FUNCTION_BLOCK FB_EP7402_Scan_Motor
VAR CONSTANT
	cnValueChannel_1: UINT:=16#8007;
	cnValueChannel_2: UINT:=16#8017;
END_VAR
VAR_INPUT
	bExecute:BOOL;
	sNetId 		: T_AmsNetID;
	tUpdateInterval:TIME:=T#1S;
	nSlaveAddr	: UINT;
	bMotorChannel_1:BOOL:= TRUE;
END_VAR
VAR_OUTPUT
	bBusy:BOOL;
	nProgress: USINT;
	aResponse:ARRAY [1..6] OF BYTE;
	bError:BOOL;
	nErrId:UDINT;
END_VAR
VAR
	fbWriteCoEParameter	:  FB_EcCoESdoWrite;
	fbReadCoEParameter	:  FB_EcCoESdoRead;
	fbReadCoEParameterEx	:  FB_EcCoESdoReadEx;
	fbRequestProgress:f_trig;
	nStep:(init, request_command_register, requesting_command_register ,send_request, sending_request, request_progress, requesting_progress, request_error, requesting_error);
	fbExecuteTrigger:r_trig;
	nStatus:USINT;
	aBuffer: array [1..12] of Byte;
	
END_VAR

fbExecuteTrigger(clk:=bExecute);
IF fbExecuteTrigger.q THEN
	nStep:=request_command_register;
	nProgress:=0;
	memset(ADR(aResponse),0,SIZEOF(aResponse));
	bBusy:=TRUE;
END_IF



CASE nStep OF
	init:
		bBusy := FALSE;
	
	request_command_register:
		fbReadCoEParameterEx(bExecute:=FALSE);
		IF NOT fbReadCoEParameterEx.bBusy THEN
			fbReadCoEParameterEx(
				sNetId:= sNetId, 
				nSlaveAddr:= nSlaveAddr, 
				nIndex:= 16#FB00, 
				pDstBuf:= ADR(aBuffer), 
				cbBufLen:= SIZEOF(aBuffer), 
				bExecute:= TRUE,
				bCompleteAccess:= TRUE,
				bError=>bError , 
				nErrId=> nErrId);
			nStep:=	requesting_command_register;
		END_IF

		
	requesting_command_register:
		fbReadCoEParameterEx(bExecute:=FALSE);
		IF NOT fbReadCoEParameterEx.bBusy THEN
			IF fbReadCoEParameterEx.bError THEN
				nStep:= init;
			ELSE
				nStep:= send_request;
			END_IF
		END_IF
		
	send_request:
		fbWriteCoEParameter(bExecute:=FALSE);
		IF NOT fbWriteCoEParameter.bBusy THEN
			fbWriteCoEParameter(
				sNetId:= sNetId, 
				nSlaveAddr:=nSlaveAddr , 
				nSubIndex:= 16#1, 
				nIndex:= 16#FB00, 
				pSrcBuf:= SEL(bMotorChannel_1, ADR(cnValueChannel_2), ADR(cnValueChannel_1)), 
				cbBufLen:= SEL(bMotorChannel_1, SIZEOF(cnValueChannel_2), SIZEOF(cnValueChannel_1)),
				bExecute:= TRUE ,
				tTimeout:= ,  
				bError=>bError , 
				nErrId=> nErrId);
			nStep:=	sending_request;
		END_IF

		
	sending_request:
		fbWriteCoEParameter(bExecute:=FALSE);
		IF NOT fbWriteCoEParameter.bBusy THEN
			IF fbWriteCoEParameter.bError THEN
				nStep:= init;
			ELSE
				nStep:= request_progress;
			END_IF
		END_IF
	
	request_progress:
		fbReadCoEParameter(bExecute:=FALSE);
		IF NOT fbReadCoEParameter.bBusy THEN
			fbReadCoEParameter(
				sNetId:= sNetId, 
				nSlaveAddr:= nSlaveAddr, 
				nSubIndex:= 16#2, 
				nIndex:= 16#FB00, 
				pDstBuf:= ADR(nStatus), 
				cbBufLen:= SIZEOF(nStatus), 
				bExecute:= TRUE,
				bError=>bError , 
				nErrId=> nErrId);
			nStep:=	requesting_progress;
		END_IF

		
	requesting_progress:
		fbReadCoEParameter(bExecute:=FALSE);
		IF NOT fbReadCoEParameter.bBusy THEN
			IF fbReadCoEParameter.bError THEN
				nStep:= init;
			ELSE
				IF nStatus>100 THEN
					nProgress:=nStatus-100;
					nStep:= request_progress;
				ELSIF nStatus=0 THEN
					nProgress:=100;
					nStep:= init;
				ELSE
					nProgress:=0;
					nStep:= request_error;					
				END_IF
			END_IF
		END_IF
		
	request_error:
		fbReadCoEParameter(bExecute:=FALSE);
		IF NOT fbReadCoEParameter.bBusy THEN
			fbReadCoEParameter(
				sNetId:= sNetId, 
				nSlaveAddr:= nSlaveAddr, 
				nSubIndex:= 16#3, 
				nIndex:= 16#FB00, 
				pDstBuf:= ADR(aResponse), 
				cbBufLen:= SIZEOF(aResponse), 
				bExecute:= TRUE,
				bError=> bError , 
				nErrId=> nErrId);
			nStep:=	requesting_error;
		END_IF

		
	requesting_error:
		fbReadCoEParameter(bExecute:=FALSE);
		IF NOT fbReadCoEParameter.bBusy THEN
				nStep:= init;
		END_IF
	
END_CASE

END_FUNCTION_BLOCK

(* stored: Version 1.1.0.1, ProductVersion 3.1.4024.12
   POU FB_EP7402_Scan_Motor: Id {5e871fc0-8447-4055-9dce-ba80d29d4a42}, SpecialFunc None *)
